{attribute addProperty BoxType "EL3403-0000-0022"}
{attribute addProperty Id "Missing_zero_crossing_AAT %I*BOOL814Missing_zero_crossing_BAT %I*BOOL815Missing_zero_crossing_CAT %I*BOOL816Phase_sequence_errorAT %I*BOOL819"}
{attribute addProperty CRC "4119957433"}
{attribute addProperty SizeInBites "32"}
{attribute addProperty SizeInBytes "4"}
TYPE PM_Status_data_F5918FB9 :
STRUCT
	{attribute addProperty Name "Missing_zero_crossing_A"}
	Missing_zero_crossing_A AT %I* : BOOL;
	{attribute addProperty Name "Missing_zero_crossing_B"}
	Missing_zero_crossing_B AT %I* : BOOL;
	{attribute addProperty Name "Missing_zero_crossing_C"}
	Missing_zero_crossing_C AT %I* : BOOL;
	{attribute addProperty Name "Phase_sequence_error"}
	Phase_sequence_error AT %I* : BOOL;
END_STRUCT
END_TYPE

(* stored: Version 1.2.0.0, ProductVersion 3.1.4024.9
   DUT PM_Status_data_F5918FB9: Id {d2b3356d-4145-49dc-9568-947c36bbe8bd} *)
